FUNCTION_BLOCK ReworkInstructionTask EXTENDS TcoCore.TcoRemoteTask
VAR
	_data:ReworkData;
END_VAR

SUPER^();

PROPERTY Data : REFERENCE TO ReworkData
GET
Data ref= _data;
END_GET
END_PROPERTY

METHOD Run : REFERENCE TO ReworkInstructionTask
VAR_INPUT
	inEntityId:STRING;
END_VAR
_data.EntityId:=inEntityId;
Run REF= THIS^;
END_METHOD

END_FUNCTION_BLOCK

(* stored: Version 1.1.0.1
   POU ReworkInstructionTask: Id {3ef14e60-716c-4442-a5d9-2c2bffc56045}, SpecialFunc None
   Property Data: Id {32b6d340-2bfe-4579-a993-a9b7903ce5f3}
   Get Get: Id {6b950daa-f7da-454b-8ac3-6244534c7457}
   Method Run: Id {dea1cab6-aaae-41ee-91e0-076daafab7df} *)
